// TwinCAT 3 PLC project Untitled1
// ProgramVersion: 3.1.4024.0
// libraries:
//   Tc2_SerialCom, * (Beckhoff Automation GmbH)
//   Tc2_Standard, * (Beckhoff Automation GmbH)
//   Tc2_System, * (Beckhoff Automation GmbH)
//   Tc3_Module, * (Beckhoff Automation GmbH)
// project tree:
//   DUTs/ ComState.TcDUT
//   / PlcTask.TcTTO
//   POUs/ MAIN.TcPOU
// real-time tasks:
//   TASK PlcTask: cycle T#10ms, priority 20, ADS port 350
// I/O:
//   DEVICE Device 3 (EtherCAT), AmsNetId 5.94.205.148.4.1
//     Term 1 (EK1100) [EK1100 EtherCAT Coupler (2A E-Bus)]
//       Term 2 (EL6021) [EL6021 Interface (RS422/485)]
//       Term 3 (EL9011) [EL9011 End Terminal]
//   DEVICE Device 2 (COM Port)
// variable links:
//   Untitled1/Untitled1 Instance <-> Device 3 (EtherCAT)/Term 1 (EK1100)/Term 2 (EL6021)
//     PlcTask Inputs/MAIN.Bf <-> COM TxPDO-Map Input 98 Byte/Buffer full
//     PlcTask Inputs/MAIN.Fe <-> COM TxPDO-Map Input 98 Byte/Framing error
//     PlcTask Inputs/MAIN.Ia <-> COM TxPDO-Map Input 98 Byte/Init accepted
//     PlcTask Inputs/MAIN.Il <-> COM TxPDO-Map Input 98 Byte/Input length
//     PlcTask Inputs/MAIN.Oe <-> COM TxPDO-Map Input 98 Byte/Overrun error
//     PlcTask Inputs/MAIN.Pe <-> COM TxPDO-Map Input 98 Byte/Parity error
//     PlcTask Inputs/MAIN.Rr <-> COM TxPDO-Map Input 98 Byte/Receive request
//     PlcTask Inputs/MAIN.RxBuffer/Buffer[{0..21}] <-> COM TxPDO-Map Input 98 Byte/Data In {0..21}  (22 links)
//     PlcTask Inputs/MAIN.Ta <-> COM TxPDO-Map Input 98 Byte/Transmit accepted
//     PlcTask Outputs/MAIN.Ir <-> COM RxPDO-Map Output 98 Byte/Init request
//     PlcTask Outputs/MAIN.Ol <-> COM RxPDO-Map Output 98 Byte/Output length
//     PlcTask Outputs/MAIN.Ra <-> COM RxPDO-Map Output 98 Byte/Receive accepted
//     PlcTask Outputs/MAIN.Sc <-> COM RxPDO-Map Output 98 Byte/Send continues
//     PlcTask Outputs/MAIN.Tr <-> COM RxPDO-Map Output 98 Byte/Transmit request
//     PlcTask Outputs/MAIN.TxBuffer/Buffer[0] <-> COM RxPDO-Map Output 98 Byte/Data Out 0
//     PlcTask Outputs/MAIN.TxBuffer/Buffer[1] <-> COM RxPDO-Map Output 98 Byte/Data Out 1

CONFIGURATION Untitled1
    RESOURCE PLC ON TwinCAT3
        TASK PlcTask(INTERVAL := T#10ms, PRIORITY := 20);
        PROGRAM MAIN WITH PlcTask : MAIN;
    END_RESOURCE
END_CONFIGURATION

// ---- DUTs/ComState.TcDUT
{attribute 'qualified_only'}
{attribute 'strict'}
TYPE ComState :
(
	Idle, Send, Recv, Process, WaitForReceive, WaitForTransmit, WaitForInit, WaitForNotInit, ClearBuffer, RecvSetUp
);
END_TYPE

// ---- POUs/MAIN.TcPOU
PROGRAM MAIN
VAR	
	TxD : ARRAY[0..1] OF BYTE;
	OKIA : BOOL := FALSE;
	OKTA : BOOL := FALSE;
	RxD : ARRAY[0..255] OF BYTE;
	State : ComState := ComState.Idle;
	SendD : SendData;
	ReceiveD : ReceiveData;
	TxBuffer AT %Q* : ComBuffer;
	RxBuffer AT %I* : ComBuffer;
	LatestValue AT %I* : BYTE;
	Status AT %I*: UINT;
	Ta AT %I* : BOOL;
	Rr AT %I* : BOOL;
	Ia AT %I* : BOOL;
	Bf AT %I* : BOOL;
	Pe AT %I* : BOOL;
	Fe AT %I* : BOOL;
	Oe AT %I* : BOOL;
	Il AT %I* : USINT;
	Tr AT %Q*: BOOL;
	Ra AT %Q*: BOOL;
	Ir AT %Q*: BOOL;
	Sc AT %Q*: BOOL;
	Ol AT %Q* : USINT;
	SCounter : INT; 
	RCounter : INT := 0;
	I : INT;
	OldRR : BOOL := Rr;
	FbClearBuffer  : ClearComBuffer;
	RxData : ARRAY[0..21] OF BYTE;
	FBRecv : ReceiveData;
	LatestReading : BYTE;
	//OldRa : BOOL;
END_VAR

(**Ignore all variables and states that don't appear in the code
Please make a new branch before writing any modifications*)

CASE State OF
	
	ComState.Idle: //Idle state, the algorithm begins here
	
		
		Ir := TRUE; //Set Init request to true
		State := ComState.WaitForInit; //wait for init accepted
	
	ComState.WaitForInit:
	
		IF Ia THEN //if init accepted turns true
			Ir := FALSE; //revert the request
			State := ComState.WaitForNotInit; //wait for init to be inverted
		END_IF
	
	ComState.WaitForNotInit:

		IF NOT Ia THEN //init inverted
			State := ComState.Send; //go to send state
		END_IF	
	
	ComState.Send:
	
		Ol := 2; //output length = 2 (length of request is 2 bytes)
		TxBuffer.Buffer[0] := 16#01; //first byte (sensor's address)
		TxBuffer.Buffer[1] := 16#87; //second byte (data stream request)
		Tr := TRUE; //set Transmission Request to true
		SCounter := SCounter + 1;
		State := ComState.WaitForTransmit; //wait for Transmission to be accepted by terminal
		
	ComState.WaitForTransmit:
		IF Ta THEN //Transmission accepted
			State := ComState.WaitForReceive; //wait for readings
		END_IF
		
	ComState.WaitForReceive:
		
		IF NOT Rr = OldRR THEN //Receive Request inverted means new data available
			OldRR := Rr; //keep track of old value
			Ra := TRUE;	//accept the receive request
			State := ComState.RecvSetUp; //set up the receive function block
		END_IF
		
	ComState.RecvSetUp:
	
		FBRecv(
			pReceiveData := ADR(RxData), //pointer to where data should go
			SizeReceiveData := SIZEOF(RxData), 
			RXbuffer := RxBuffer //buffer where data is received
		);
		State := ComState.Recv;
	ComState.Recv:
	
		IF FBRecv.DataReceived THEN
			ADSLOGSTR(msgCtrlMask := ADSLOG_MSGTYPE_ERROR OR ADSLOG_MSGTYPE_LOG,
				msgFmtStr := 'Log %s',
				strArg := 'Data received');
			LatestReading := RxData[21];
			State := ComState.WaitForReceive; //wait for new data
		END_IF
				
END_CASE

END_PROGRAM
